FUNCTION_BLOCK PixelWritter EXTENDS FB_CyclicFB IMPLEMENTS ITF_PixelWritter
VAR
	CtrlOut AT %Q*: Control;
	StatusIn AT %I*: Status;
	ExtCtrlOut AT %Q*: ExtendedControl;
	UpdateRTrig: R_TRIG;
	UpdateFTrig: F_TRIG;
	ClearPixels: BOOL;
END_VAR

METHOD ClearPixelArrayCommand : BOOL
IF NOT ClearPixels THEN
	CtrlOut.PixelCommand.Command := 2;
	CtrlOut.Execute := NOT CtrlOut.Execute;
END_IF
END_METHOD

METHOD CyclicLogic : BOOL
SUPER^.CyclicLogic();
UpdateFTrig(CLK := StatusIn.UpdateAck);
UpdateRTrig(CLK := StatusIn.UpdateAck);
IF UpdateFTrig.Q OR UpdateRTrig.Q THEN
	CtrlOut.Update := FALSE;
	ExtCtrlOut.Update := FALSE;
END_IF
END_METHOD

METHOD ForwardCommandToFrameBuffer : BOOL
IF NOT ForwardCommandToFrameBuffer THEN
	CtrlOut.Execute := NOT CtrlOut.Execute;
	CtrlOut.Update := TRUE;
	ForwardCommandToFrameBuffer := TRUE;
END_IF
END_METHOD

METHOD ForwardExtCommandToFrame : BOOL
IF NOT ForwardExtCommandToFrame THEN
	ExtCtrlOut.Execute := NOT ExtCtrlOut.Execute;
	ExtCtrlOut.Update := TRUE;
	ExtCtrlOut.Write := FALSE;
	ForwardExtCommandToFrame := TRUE;
END_IF
END_METHOD

METHOD SendCommandToPixelBuffer : BOOL
VAR_INPUT
	NewCommand: Command;
END_VAR
IF NOT StatusIn.Busy THEN
	SendCommandToPixelBuffer := TRUE;
	CtrlOut.PixelCommand := NewCommand;
	CtrlOut.Execute := NOT CtrlOut.Execute;
END_IF
END_METHOD

METHOD SendExtCommand : BOOL
VAR_INPUT
	NewCommand: ExtendedCommand;
END_VAR
IF NOT StatusIn.Busy THEN
	SendExtCommand := TRUE;
	ExtCtrlOut.Command := NewCommand;
	ExtCtrlOut.Write := TRUE;
	ExtCtrlOut.Execute := NOT ExtCtrlOut.Execute;
END_IF
END_METHOD

END_FUNCTION_BLOCK

(* stored: Version 1.1.0.1, ProductVersion 3.1.4024.13
   POU PixelWritter: Id {059a66e7-2117-4fdc-9a96-c27b3bb8a014}, SpecialFunc None
   Method ClearPixelArrayCommand: Id {da74ea2f-483d-49f6-a01a-d07fa5a3e740}
   Method CyclicLogic: Id {411f79cb-7bfe-4944-9b09-24abdc0e156c}
   Method ForwardCommandToFrameBuffer: Id {401ed8b0-49c7-4044-ad85-4e6fc03f46a0}
   Method ForwardExtCommandToFrame: Id {838d00e5-96fb-4eea-a1a4-d84527e6f813}
   Method SendCommandToPixelBuffer: Id {d6b8d03d-e674-46aa-9859-7a3d82607b1a}
   Method SendExtCommand: Id {bded14ba-ba3e-4bb4-ba01-208d5142a337} *)
